(* Schneider Machine Expert - Basic project Exercise-8- Using Memory as Latch, file version 2.9.0.0 *)
(* ProjectInformations: Name=New project *)

HARDWARE
  Cpu 0: TM221CE24R
  EthernetConfiguration: NetworkName=M221, IpAllocationMode=FixedAddress, IpAddress=0.0.0.0, SubnetMask=0.0.0.0
  SerialLineConfiguration: Baud=Baud19200, Parity=ParityEven, DataBits=DataBits8, StopBits=StopBits1, PhysicalMedium=PhysicalMediumRs485, SlaveId=1, Addressing=SlaveAddressing
  MastTask: UsePeriodScanMode=false, PeriodScan=100
  FastTask: Period=255
  CpuBehavior: StartingMode=StartAsPreviousState, AutoSaveRamOnEeprom=true, WatchdogPeriod=250

SYMBOLS  (address, symbol, comment, settings)
  %M0       MEMORY_1
  %M1       MEMORY_2
  %I0.0     SWITCH_1
  %I0.1     SWITCH_2
  %I0.2     SWITCH_3
  %Q0.0     LED_1
  %Q0.1     LED_2
  %Q0.2     LED_3
  %Q0.3     LED_4

POU New POU
  (* SectionNumber=1 *)

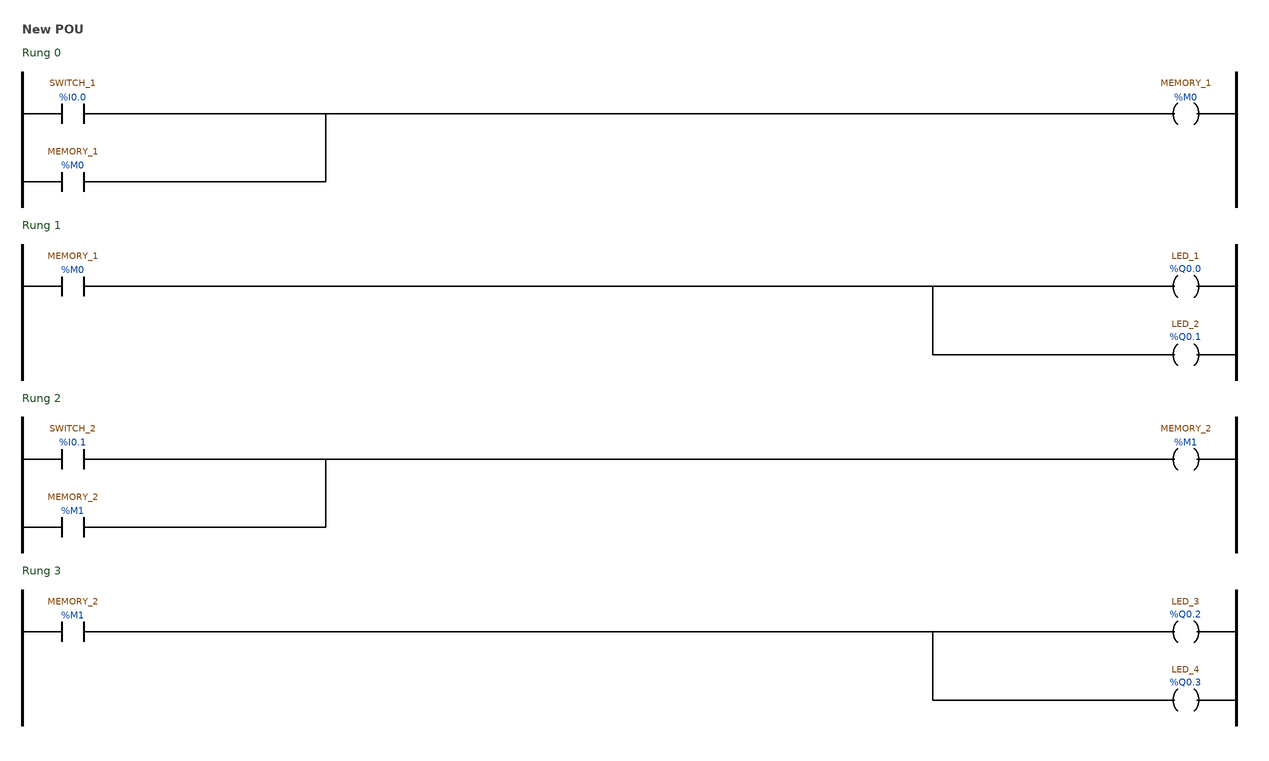

// Rung 0
  LD %I0.0                (* SWITCH_1 *)
  OR %M0                  (* MEMORY_1 *)
  ST %M0                  (* MEMORY_1 *)
  // as ST:
  //   MEMORY_1 := SWITCH_1 OR MEMORY_1;

// Rung 1
  LD %M0                  (* MEMORY_1 *)
  ST %Q0.0                (* LED_1 *)
  ST %Q0.1                (* LED_2 *)
  // as ST:
  //   LED_1 := MEMORY_1;
  //   LED_2 := MEMORY_1;

// Rung 2
  LD %I0.1                (* SWITCH_2 *)
  OR %M1                  (* MEMORY_2 *)
  ST %M1                  (* MEMORY_2 *)
  // as ST:
  //   MEMORY_2 := SWITCH_2 OR MEMORY_2;

// Rung 3
  LD %M1                  (* MEMORY_2 *)
  ST %Q0.2                (* LED_3 *)
  ST %Q0.3                (* LED_4 *)
  // as ST:
  //   LED_3 := MEMORY_2;
  //   LED_4 := MEMORY_2;
